FUNCTION_BLOCK FB_DeurSensor IMPLEMENTS ITF_DeurSensor
VAR_INPUT
	I_DeurSensorOpen : BOOL; // OPEN = TRUE, DICHT = FALSE
END_VAR

PROPERTY DeurSensorOpen : BOOL
GET
DeurSensorOpen := I_DeurSensorOpen;
END_GET
END_PROPERTY

END_FUNCTION_BLOCK

(* stored: Version 1.1.0.1
   POU FB_DeurSensor: Id {5666ae5d-de79-43ff-927a-d72f98f4a42f}, SpecialFunc None
   Folder Properties: Id {591b7c54-2b61-4540-b499-8e77d1f36dbc}
   Property DeurSensorOpen: Id {6eb3df85-7518-4e87-8f15-a36aab9be3a5}
   Get Get: Id {8ed1b79f-02cc-4a3b-ac79-9c11d2e8a2f3} *)
